% RSLogix 500 project PIRU HEATED FLOODER LEMON LINE_BAK002.RSS, saved by version 11.00.00.00 %
PROJECT "UNTITLED"    % processor: MicroLogix 1200 %

PROGRAM FILES
  LAD 2   13 rungs

DATA FILES
  O0 OUTPUT  4 elements
  I1 INPUT  4 elements
  S2 STATUS  66 elements
  B3 BINARY  1 elements
  T4 TIMER  1 elements
  C5 COUNTER  1 elements
  R6 CONTROL  1 elements
  N7 INTEGER  1 elements
  F8 FLOAT  1 elements

LADDER 2
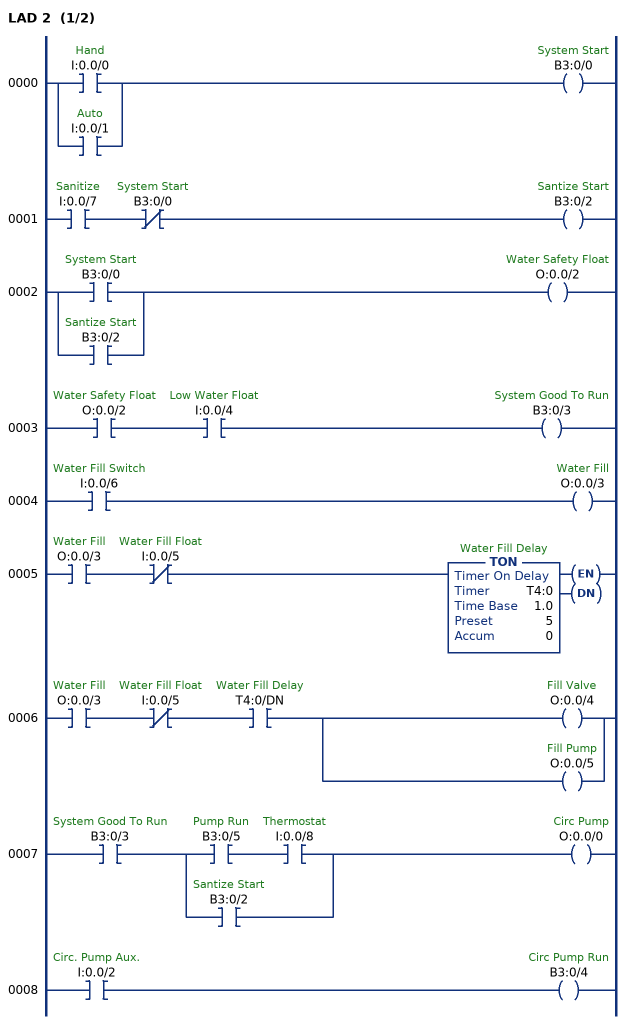
% Rung: 0 %
SOR BST XIC I:0.0/0 NXB XIC I:0.0/1 BND OTE B3:0/0 EOR
%   I:0.0/0  "Hand" %
%   I:0.0/1  "Auto" %
%   B3:0/0  "System Start" %
% Rung: 1 %
SOR XIC I:0.0/7 XIO B3:0/0 OTE B3:0/2 EOR
%   I:0.0/7  "Sanitize" %
%   B3:0/0  "System Start" %
%   B3:0/2  "Santize Start" %
% Rung: 2 %
SOR BST XIC B3:0/0 NXB XIC B3:0/2 BND OTE O:0.0/2 EOR
%   B3:0/0  "System Start" %
%   B3:0/2  "Santize Start" %
%   O:0.0/2  "Water Safety Float" %
% Rung: 3 %
SOR XIC O:0.0/2 XIC I:0.0/4 OTE B3:0/3 EOR
%   O:0.0/2  "Water Safety Float" %
%   I:0.0/4  "Low Water Float" %
%   B3:0/3  "System Good To Run" %
% Rung: 4 %
SOR XIC I:0.0/6 OTE O:0.0/3 EOR
%   I:0.0/6  "Water Fill Switch" %
%   O:0.0/3  "Water Fill" %
% Rung: 5 %
SOR XIC O:0.0/3 XIO I:0.0/5 TON T4:0 1.0 5 0 EOR
%   O:0.0/3  "Water Fill" %
%   I:0.0/5  "Water Fill Float" %
%   T4:0  "Water Fill Delay" %
% Rung: 6 %
SOR XIC O:0.0/3 XIO I:0.0/5 XIC T4:0/DN BST OTE O:0.0/4 NXB OTE O:0.0/5 BND EOR
%   O:0.0/3  "Water Fill" %
%   I:0.0/5  "Water Fill Float" %
%   T4:0  "Water Fill Delay" %
%   O:0.0/4  "Fill Valve" %
%   O:0.0/5  "Fill Pump" %
% Rung: 7 %
SOR XIC B3:0/3 BST XIC B3:0/5 XIC I:0.0/8 NXB XIC B3:0/2 BND OTE O:0.0/0 EOR
%   B3:0/3  "System Good To Run" %
%   B3:0/5  "Pump Run" %
%   I:0.0/8  "Thermostat" %
%   B3:0/2  "Santize Start" %
%   O:0.0/0  "Circ Pump" %
% Rung: 8 %
SOR XIC I:0.0/2 OTE B3:0/4 EOR
%   I:0.0/2  "Circ. Pump Aux." %
%   B3:0/4  "Circ Pump Run" %

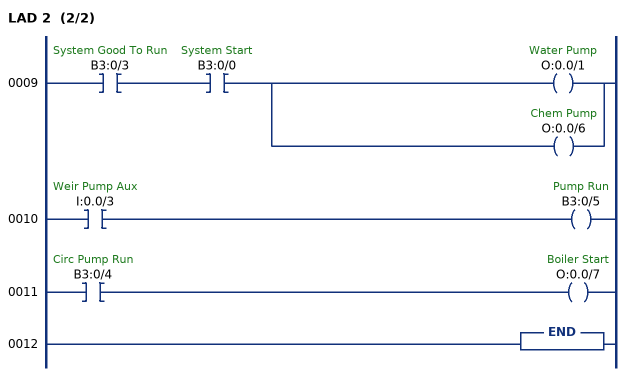
% Rung: 9 %
SOR XIC B3:0/3 XIC B3:0/0 BST OTE O:0.0/1 NXB OTE O:0.0/6 BND EOR
%   B3:0/3  "System Good To Run" %
%   B3:0/0  "System Start" %
%   O:0.0/1  "Water Pump" %
%   O:0.0/6  "Chem Pump" %
% Rung: 10 %
SOR XIC I:0.0/3 OTE B3:0/5 EOR
%   I:0.0/3  "Weir Pump Aux" %
%   B3:0/5  "Pump Run" %
% Rung: 11 %
SOR XIC B3:0/4 OTE O:0.0/7 EOR
%   B3:0/4  "Circ Pump Run" %
%   O:0.0/7  "Boiler Start" %
% Rung: 12 %
SOR END EOR

DATA TABLE (non-zero values as saved)
DATA B3
% B3:0 % 0X0039
DATA T4
% .PRE .ACC %
% T4:0 % 5 0
